{attribute 'qualified_only'}
VAR_GLOBAL
END_VAR

(* stored: Version 1.1.0.1, ProductVersion 3.1.4022.18
   GVL GVL_CryoStat: Id {3975b31a-b7d4-48c4-bd57-f1035c11169e} *)
